Universal Robots PolyScope program: lab 3 mike .urp

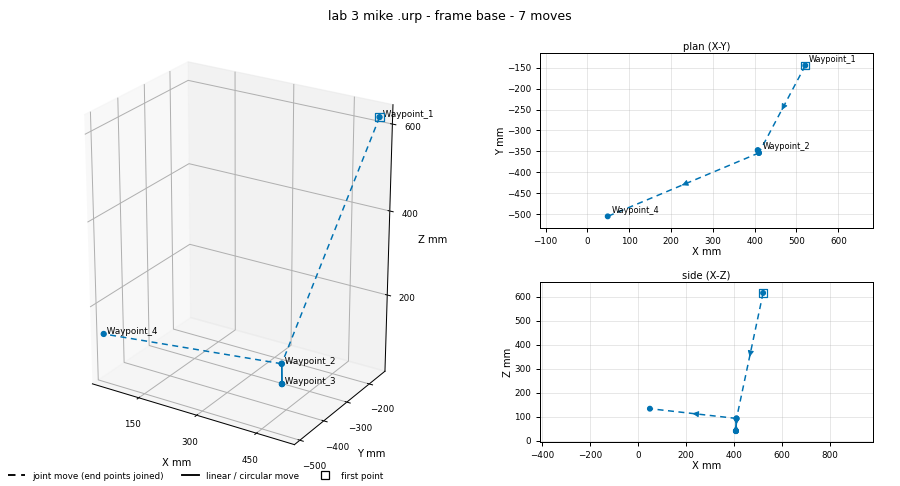
[picture p0: tool path of lab 3 mike .urp in frame base, 7 of 7 moves have a stored position in this frame; points joined in program order, loops and branches not executed]
Program lab 3 mike  (installation=default directory=/programs createdIn=5.14.5 lastSavedIn=5.14.5 robotSerialNumber=20195300809)
Calibrated DH parameters: a=[-0.000085, -0.20076, -0.212369, 0.000121, -0.000118, 0]; d=[0.15185, -26.306375, 24.753047, 1.684739, 0.085386, 0.092088]; alpha=[1.572149, -0.00522, -0.011864, 1.571339, -1.571085, 0]; deltaTheta=[0, 0.599885, -0.513355, -0.086555, 0.000006, 0]
InitVariablesNode
Robot Program (runOnlyOnce=false)
  MoveJ speed 60 deg/s, acceleration 80 deg/s^2 (useActiveTCP=true) feature=Base
    Waypoint Waypoint_1: TCP in base x=521.017 y=-144.678 z=616.617 mm, rx=-0.7391 ry=0.9171 rz=-1.5297 rad; joints [137.978, -49.137, 24.923, -189.355, -62.369, 18.525] deg; TCP offset x=0 y=0 z=150 mm, rx=0 ry=0 rz=0 rad
    URCap Gripper (Robotiq_Grippers, Robotiq Inc.) dataModel(position=0.0, force=0.0, speed=0.0, positionInDouble=0.0, forceInDouble=0.0, speedInDouble=0.0, slaveIds=[9], blocking=true)
    Popup Message (haltProgram=false message=give me the patch please  inputType=Text)
    URCap Gripper (Robotiq_Grippers, Robotiq Inc.) dataModel(position=100.0, force=0.0, speed=0.0, positionInDouble=100.0, forceInDouble=0.0, speedInDouble=0.0, slaveIds=[9], blocking=true)
    MoveJ speed 60 deg/s, acceleration 80 deg/s^2 (useActiveTCP=true) feature=Base
      Waypoint Waypoint_2: TCP in base x=410.192 y=-353.673 z=92.897 mm, rx=-0.1665 ry=3.107 rz=-0.1571 rad; joints [126.12, -29.309, 15.086, -81.461, -92.787, 29.855] deg
    MoveL speed 250 mm/s, acceleration 1200 mm/s^2 (useActiveTCP=true) feature=Base
      Waypoint Waypoint_3: TCP in base x=408.096 y=-347.954 z=40.684 mm, rx=0.1685 ry=-3.1209 rz=0.0339 rad; joints [126.106, -23.617, 15.359, -82.3, -92.341, 29.861] deg
    MoveJ speed 60 deg/s, acceleration 80 deg/s^2 (useActiveTCP=true) feature=Base
      Waypoint Waypoint_5: TCP in base x=408.073 y=-347.972 z=40.686 mm, rx=0.1685 ry=-3.1208 rz=0.0339 rad; joints [126.104, -23.618, 15.358, -82.299, -92.343, 29.86] deg; TCP offset x=0 y=0 z=150 mm, rx=0 ry=0 rz=0 rad
    MoveJ speed 60 deg/s, acceleration 80 deg/s^2 (useActiveTCP=true) feature=Base
      Waypoint Waypoint_6: TCP in base x=407.178 y=-347.13 z=39.66 mm, rx=2.7986 ry=-1.3709 rz=-0.0137 rad; joints [126.108, -23.585, 15.443, -82.103, -92.407, -91.754] deg; TCP offset x=0 y=0 z=150 mm, rx=0 ry=0 rz=0 rad
    MoveL speed 250 mm/s, acceleration 1200 mm/s^2 (useActiveTCP=true) feature=Base
      Waypoint Waypoint_2: TCP in base x=410.192 y=-353.673 z=92.897 mm, rx=-0.1665 ry=3.107 rz=-0.1571 rad; joints [126.12, -29.309, 15.086, -81.461, -92.787, 29.855] deg; TCP offset x=0 y=0 z=150 mm, rx=0 ry=0 rz=0 rad
    MoveJ speed 60 deg/s, acceleration 80 deg/s^2 (useActiveTCP=true) feature=Base
      Waypoint Waypoint_4: TCP in base x=48.589 y=-505.342 z=133.6 mm, rx=-0.013 ry=3.0065 rz=-0.8991 rad; joints [76.745, -69.226, 94.44, -147.685, -82.991, -12.129] deg
    Force Frame feature=Plane_1; selection=[1, 1, 0, 0, 0, 0]; wrench=[0, 0, 0, 0, 0, 0]; limitsForce=[0.15, 0.15, 0.15, 1.047198, 1.047198, 1.047198]; limitsMotion=[0.1, 0.1, 0.1, 0.349066, 0.349066, 0.349066]
      Popup Message (haltProgram=false message=position patch inputType=Text)
    Force Frame feature=Plane_1; selection=[0, 0, 1, 0, 0, 0]; wrench=[0, 0, -5, 0, 0, 0]; limitsForce=[0.15, 0.15, 0.15, 1.047198, 1.047198, 1.047198]; limitsMotion=[0.1, 0.1, 0.1, 0.349066, 0.349066, 0.349066]
      Wait Sleep waitTime=5
      URCap Gripper (Robotiq_Grippers, Robotiq Inc.) dataModel(position=0.0, force=0.0, speed=0.0, positionInDouble=0.0, forceInDouble=0.0, speedInDouble=0.0, slaveIds=[9], blocking=true)
    MoveL speed 250 mm/s, acceleration 1200 mm/s^2 (useActiveTCP=true) feature=Plane_1
      MoveDirectionNode (selectedDirection=ZPlus) feature(featureName=Plane_1)
        Until DISTANCE (allowActions=false deceleration=3 distanceNodeType=STOP) Distance=0.1; motionParameters(blendRadius=0)
    Popup Message (haltProgram=false message=patch stuck! inputType=Text)
